{attribute 'pack_mode' := '1'}
TYPE TVacuumSettingsMMI :
STRUCT
	TTable				: TVaccumSettings;
	TLoaderHead		: TVaccumSettings;
	TLoaderPlate			: TVaccumSettings;
	TTurnOver			: TVaccumSettings;
	iTablePartialDelay	: INT;
END_STRUCT
END_TYPE

(* stored: Version 1.1.0.1, ProductVersion 3.1.4022.12
   DUT TVacuumSettingsMMI: Id {2299021b-7f3f-434e-8766-63f837781263} *)
